(* IEC 61131-3 sources: RL_MAR/experiments/comparison/llm4plc/results/gpt-4o-mini_20260506_100619/20260506_102845, 3 files *)

(* ---- generated_code_iteration_0.st ---- *)
ructured-text
FUNCTION_BLOCK FB_RequestHandler
VAR_IN
    request : BOOL; // Input for request signal
    done : BOOL; // Input for processing completion signal
END_VAR_IN
VAR_OUT
    listen : BOOL; // Output for listening mode
END_VAR_OUT
VAR
    state : INT := 0; // State variable initialized to 0
END_VAR

// Implement state logic in the function block
IF state = 0 THEN
    IF request = FALSE THEN
        listen := TRUE; // Set listen to TRUE and remain in STATE 0
    ELSE
        listen := FALSE; // Set listen to FALSE
        state := 1; // Transition to STATE 1
        done := FALSE; // Set done to FALSE
    END_IF
ELSIF state = 1 THEN
    IF done = FALSE THEN
        // Remain in STATE 1
    ELSE
        state := 0; // Transition back to STATE 0
        listen := TRUE; // Set listen to TRUE
    END_IF
END_IF

END_FUNCTION_BLOCK

(* ---- generated_code_iteration_1.st ---- *)
START_REASON
The errors in the original Structured Text (ST) code occurred due to the incorrect use of variable section declarations. Specifically, the code used "VAR_IN" and "VAR_OUT," which are not valid in the context of a FUNCTION_BLOCK in Structured Text. Instead, the correct sections to use are "VAR_INPUT" for input variables and "VAR_OUTPUT" for output variables. Additionally, the variable section for internal variables should simply be "VAR" and should be closed with "END_VAR."
END_REASON

START_ST
FUNCTION_BLOCK FB_RequestHandler
VAR_INPUT
    request : BOOL; // Input for request signal
    done : BOOL; // Input for processing completion signal
END_VAR_INPUT
VAR_OUTPUT
    listen : BOOL; // Output for listening mode
END_VAR_OUTPUT
VAR
    state : INT := 0; // State variable initialized to 0
END_VAR

// Implement state logic in the function block
IF state = 0 THEN
    IF request = FALSE THEN
        listen := TRUE; // Set listen to TRUE and remain in STATE 0
    ELSE
        listen := FALSE; // Set listen to FALSE
        state := 1; // Transition to STATE 1
        done := FALSE; // Set done to FALSE
    END_IF
ELSIF state = 1 THEN
    IF done = FALSE THEN
        // Remain in STATE 1
    ELSE
        state := 0; // Transition back to STATE 0
        listen := TRUE; // Set listen to TRUE
    END_IF
END_IF

END_FUNCTION_BLOCK
END_ST

(* ---- generated_code_iteration_2.st ---- *)
START_REASON
The errors in the original Structured Text (ST) code occurred due to the incorrect use of variable section declarations. Specifically, the code used "VAR_INPUT" and "VAR_OUTPUT," which are not valid in the context of a FUNCTION_BLOCK in Structured Text. The correct sections to use are "VAR" for internal variables and "VAR" for output variables, and all variable declarations should be enclosed within a single "VAR" section. Additionally, the variable section should be closed with "END_VAR."
END_REASON

START_ST
FUNCTION_BLOCK FB_RequestHandler
VAR
    request : BOOL; // Input for request signal
    done : BOOL; // Input for processing completion signal
    listen : BOOL; // Output for listening mode
    state : INT := 0; // State variable initialized to 0
END_VAR

// Implement state logic in the function block
IF state = 0 THEN
    IF request = FALSE THEN
        listen := TRUE; // Set listen to TRUE and remain in STATE 0
    ELSE
        listen := FALSE; // Set listen to FALSE
        state := 1; // Transition to STATE 1
        done := FALSE; // Set done to FALSE
    END_IF
ELSIF state = 1 THEN
    IF done = FALSE THEN
        // Remain in STATE 1
    ELSE
        state := 0; // Transition back to STATE 0
        listen := TRUE; // Set listen to TRUE
    END_IF
END_IF

END_FUNCTION_BLOCK
END_ST
